ABB RobotStudio station: Solution1_Hicham.rspag

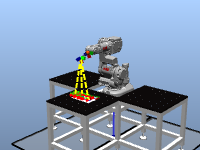
--- station ---
Station Solution1_Hicham (saved by RobotStudio 7.0.8504.151)
Controller IRB_140_6kg_0.81m, task T_ROB1: task frame (RAPID world) sits at (0, 0, 670) mm in the station
Controller IRB_140_6kg_0.81m
  mechanical unit ROB_1: IRB140_6_81_C_03, 6 joints, base frame (0, 0, 0) mm
Layout (positions relative to the parent item):
  - IRB140_6_81_C_03 [mechanism, from Robots\IRB140_6_81_C_G_03.rslib] at (0, 0, 670) mm; joint values [0, 0, 0, 0, 0.2618, 0] (rad or m)
  - rob-table [part, from Libraries\rob-table.rslib]
  - pen [mechanism, from Libraries\pen.rslib] at (512.79, 0, 1365.18) mm, rotated rx -180 ry 75 rz -180 deg
  - paper [part, from Libraries\paper.rslib]
Attachment: pen is attached to IRB140_6_81_C_03 / Link6
Targets, tools, work objects and paths stored in the station and not in the controller backup, written as RAPID:
! task T_ROB1
MODULE Module1
  CONST robtarget Target_E_10:=[[100,270,0],[1,0,0,0],[0,0,0,0],[9E+09,9E+09,9E+09,9E+09,9E+09,9E+09]];
  CONST robtarget Target_E_20:=[[100,220,0],[1,0,0,0],[-1,0,1,0],[9E+09,9E+09,9E+09,9E+09,9E+09,9E+09]];
  CONST robtarget Target_E_30:=[[50,220,0],[1,0,0,0],[-1,0,1,0],[9E+09,9E+09,9E+09,9E+09,9E+09,9E+09]];
  CONST robtarget Target_E_40:=[[0,220,0],[1,0,0,0],[-1,0,1,0],[9E+09,9E+09,9E+09,9E+09,9E+09,9E+09]];
  CONST robtarget Target_E_50:=[[0,270,0],[1,0,0,0],[-1,0,1,0],[9E+09,9E+09,9E+09,9E+09,9E+09,9E+09]];
  CONST robtarget Target_E_60:=[[50,270,0],[1,0,0,0],[-1,0,1,0],[9E+09,9E+09,9E+09,9E+09,9E+09,9E+09]];
  PROC Path_E()
    MoveL Target_E_10,v1000,z100,pen\WObj:=Workobject_1;
    MoveL offs(Target_E_10,0,0,15),v100,z1,pen\WObj:=Workobject_1;
    MoveL offs(Target_E_20,0,0,15),v100,z1,pen\WObj:=Workobject_1;
    MoveL offs(Target_E_40,0,0,15),v100,z1,pen\WObj:=Workobject_1;
    MoveL offs(Target_E_50,0,0,15),v100,z1,pen\WObj:=Workobject_1;
    MoveL offs(Target_E_30,0,0,15),v100,z1,pen\WObj:=Workobject_1;
    MoveL offs(Target_E_60,0,0,15),v100,z1,pen\WObj:=Workobject_1;
    MoveL Target_E_60,v1000,z100,pen\WObj:=Workobject_1;
    MoveJ Target_10,v1000,z100,pen\WObj:=wobj0;
  ENDPROC
ENDMODULE


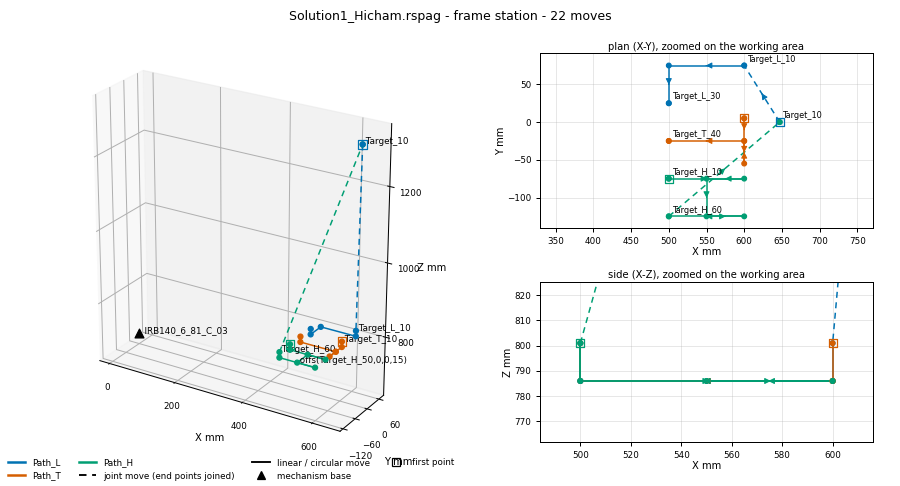
[picture p0: tool path of Solution1_Hicham.rspag in frame station, 22 of 22 moves have a stored position in this frame; points joined in program order, loops and branches not executed]
--- Backups/IRB_140_6kg_0.81m/RAPID/TASK1/PROGMOD/CalibData.mod ---
MODULE CalibData
    PERS tooldata pen:=[TRUE,[[0,0,139],[1,0,0,0]],[0.5,[0,0,20],[1,0,0,0],0,0,0]];
	TASK PERS wobjdata Workobject_1:=[FALSE,TRUE,"",[[450,125,116],[0,1,0,0]],[[50,50,-15],[1,0,0,0]]];

ENDMODULE

--- Backups/IRB_140_6kg_0.81m/RAPID/TASK1/PROGMOD/Module1.mod ---
MODULE Module1
	CONST robtarget Target_L_10:=[[100,0,0],[1,0,0,0],[0,0,-2,0],[9E+09,9E+09,9E+09,9E+09,9E+09,9E+09]];
	CONST robtarget Target_L_20:=[[0,0,0],[1,0,0,0],[0,0,-2,0],[9E+09,9E+09,9E+09,9E+09,9E+09,9E+09]];
	CONST robtarget Target_L_30:=[[0,50,0],[1,0,0,0],[0,0,-2,0],[9E+09,9E+09,9E+09,9E+09,9E+09,9E+09]];
	CONST robtarget Target_T_10:=[[100,70,0],[1,0,0,0],[0,0,-2,0],[9E+09,9E+09,9E+09,9E+09,9E+09,9E+09]];
	CONST robtarget Target_T_20:=[[100,100,0],[1,0,0,0],[0,0,-2,0],[9E+09,9E+09,9E+09,9E+09,9E+09,9E+09]];
	CONST robtarget Target_T_30:=[[100,130,0],[1,0,0,0],[0,0,-2,0],[9E+09,9E+09,9E+09,9E+09,9E+09,9E+09]];
	CONST robtarget Target_T_40:=[[0,100,0],[1,0,0,0],[0,0,-2,0],[9E+09,9E+09,9E+09,9E+09,9E+09,9E+09]];
	CONST robtarget Target_H_10:=[[0,150,0],[1,0,0,0],[0,0,-2,0],[9E+09,9E+09,9E+09,9E+09,9E+09,9E+09]];
	CONST robtarget Target_H_20:=[[50,150,0],[1,0,0,0],[0,0,-2,0],[9E+09,9E+09,9E+09,9E+09,9E+09,9E+09]];
	CONST robtarget Target_H_30:=[[100,150,0],[1,0,0,0],[0,0,-2,0],[9E+09,9E+09,9E+09,9E+09,9E+09,9E+09]];
	CONST robtarget Target_H_40:=[[100,200,0],[1,0,0,0],[0,0,-2,0],[9E+09,9E+09,9E+09,9E+09,9E+09,9E+09]];
	CONST robtarget Target_H_50:=[[50,200,0],[1,0,0,0],[0,0,-2,0],[9E+09,9E+09,9E+09,9E+09,9E+09,9E+09]];
	CONST robtarget Target_H_60:=[[0,200,0],[1,0,0,0],[0,0,-2,0],[9E+09,9E+09,9E+09,9E+09,9E+09,9E+09]];
    CONST robtarget Target_10:=[[647.048868101,0,659.200913076],[0.608761426,-0.000000006,0.793353343,-0.000000005],[0,-1,-1,0],[9E+09,9E+09,9E+09,9E+09,9E+09,9E+09]];
!    CONST robtarget Target_E_10:=[[100,270,0],[1,0,0,0],[0,0,0,0],[9E+09,9E+09,9E+09,9E+09,9E+09,9E+09]];
!    CONST robtarget Target_E_20:=[[100,220,0],[1,0,0,0],[-1,0,1,0],[9E+09,9E+09,9E+09,9E+09,9E+09,9E+09]];
!    CONST robtarget Target_E_30:=[[50,220,0],[1,0,0,0],[-1,0,1,0],[9E+09,9E+09,9E+09,9E+09,9E+09,9E+09]];
!    CONST robtarget Target_E_40:=[[0,220,0],[1,0,0,0],[-1,0,1,0],[9E+09,9E+09,9E+09,9E+09,9E+09,9E+09]];
!    CONST robtarget Target_E_50:=[[0,270,0],[1,0,0,0],[-1,0,1,0],[9E+09,9E+09,9E+09,9E+09,9E+09,9E+09]];
!    CONST robtarget Target_E_60:=[[50,270,0],[1,0,0,0],[-1,0,1,0],[9E+09,9E+09,9E+09,9E+09,9E+09,9E+09]];
    !***********************************************************
    !
    ! Module:  Module1
    !
    ! Description:
    !   Exercise 1, Robot Studio, using a pen tool
    !   (FRTF20/MMKF15 Applied Robotics), LTH, Lund University
    !
    ! Author: Hicham Mohamad (hi8826mo-s)
    !
    ! Version: 1.0
    !
    !***********************************************************


    !***********************************************************
    !
    ! Procedure main
    !
    !   This is the entry point of your program
    !
    !***********************************************************
    PROC main()
        !Add your code here
        Path_L;
        Path_T;
        Path_H;
        !Path_E;
    ENDPROC
	PROC Path_L()
	    MoveJ Target_10,v1000,z100,pen\WObj:=wobj0; ! starting at Home position
	    MoveJ Target_L_10,v100,z5,pen\WObj:=Workobject_1; ! target outside the paper
	    MoveL offs(Target_L_10,0,0,15),v100,z1,pen\WObj:=Workobject_1;
        MoveL offs(Target_L_20,0,0,15),v100,z1,pen\WObj:=Workobject_1; ! targets inside the paper
        MoveL offs(Target_L_30,0,0,15),v100,z1,pen\WObj:=Workobject_1;
	    MoveL Target_L_30,v1000,z100,pen\WObj:=Workobject_1;
	ENDPROC
	PROC Path_T()
	    MoveL Target_T_10,v1000,z100,pen\WObj:=Workobject_1;
        MoveL offs(Target_T_10,0,0,15),v100,z1,pen\WObj:=Workobject_1;
	    MoveL offs(Target_T_20,0,0,15),v100,z1,pen\WObj:=Workobject_1;
	    MoveL offs(Target_T_30,0,0,15),v100,z1,pen\WObj:=Workobject_1;
        MoveL offs(Target_T_20,0,0,15),v100,z1,pen\WObj:=Workobject_1;
	    MoveL offs(Target_T_40,0,0,15),v100,z1,pen\WObj:=Workobject_1;
        MoveL Target_T_40,v1000,z100,pen\WObj:=Workobject_1;
	ENDPROC
	PROC Path_H()
        MoveL Target_H_10,v1000,z100,pen\WObj:=Workobject_1;
	    MoveL offs(Target_H_10,0,0,15),v100,z1,pen\WObj:=Workobject_1;
	    !MoveL offs(Target_H_20,0,0,15),v100,z1,pen\WObj:=Workobject_1;
	    MoveL offs(Target_H_30,0,0,15),v100,z1,pen\WObj:=Workobject_1;
        MoveL offs(Target_H_20,0,0,15),v100,z1,pen\WObj:=Workobject_1;
        MoveL offs(Target_H_50,0,0,15),v100,z1,pen\WObj:=Workobject_1;
	    MoveL offs(Target_H_40,0,0,15),v100,z1,pen\WObj:=Workobject_1;
	    !MoveL offs(Target_H_50,0,0,15),v100,z1,pen\WObj:=Workobject_1;
	    MoveL offs(Target_H_60,0,0,15),v100,z1,pen\WObj:=Workobject_1;
        MoveL Target_H_60,v1000,z100,pen\WObj:=Workobject_1;
        MoveJ Target_10,v1000,z100,pen\WObj:=wobj0; ! Ending at Home position
	ENDPROC
!    PROC Path_E()
!        MoveL Target_E_10,v1000,z100,pen\WObj:=Workobject_1;
!        MoveL offs(Target_E_10,0,0,15),v100,z1,pen\WObj:=Workobject_1;
!        MoveL offs(Target_E_20,0,0,15),v100,z1,pen\WObj:=Workobject_1;
!        !MoveL offs(Target_E_30,0,0,15),v100,z1,pen\WObj:=Workobject_1;
!        MoveL offs(Target_E_40,0,0,15),v100,z1,pen\WObj:=Workobject_1;
!        MoveL offs(Target_E_50,0,0,15),v100,z1,pen\WObj:=Workobject_1;
!        MoveL offs(Target_E_30,0,0,15),v100,z1,pen\WObj:=Workobject_1;
!        MoveL offs(Target_E_60,0,0,15),v100,z1,pen\WObj:=Workobject_1;
!        MoveL Target_E_60,v1000,z100,pen\WObj:=Workobject_1;
!        MoveJ Target_10,v1000,z100,pen\WObj:=wobj0; ! Ending at Home position
!    ENDPROC
ENDMODULE
